// TIA Portal V18 export
ORGANIZATION_BLOCK "Main"   // OB1, LAD, ProgramCycle
TITLE = "Main Program Sweep (Cycle)"
{ S7_Optimized_Access := 'TRUE' }
// Bonanza Elect TD Rev0
// Written By Kristopher Gimenez January 16,2023
// For any questions please contact Automated Rig Technogies @ 403-723-6602
// This program is for the control the Bonanza Top drives utlizing the electric HPU.
// stored: SetENOAutomatically false
   VAR_INPUT
      Initial_Call : Bool;   // Initial call of this OB
      Remanence : Bool;   // =True, if remanent data are available
   END_VAR
   VAR_TEMP   // added for the SCL form of the ladder/FBD networks
      _w1 : Bool;
   END_VAR
BEGIN

REGION Network 2: Comm Checks, Communication is online after control system is powered up for 1min 10s. So to check when the system is full powered up
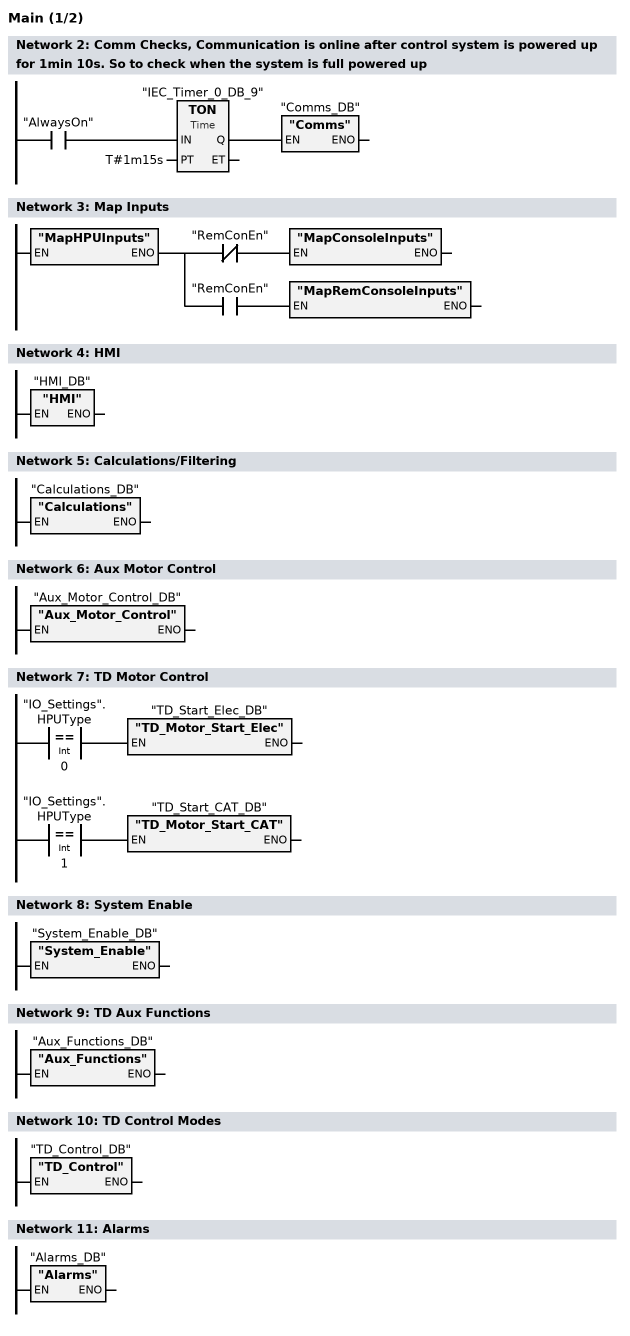
   RUNG wire#powerrail
      Contact( "AlwaysOn" )
      { S7_Templates := "time_type := Time" } "IEC_Timer_0_DB_9".TON(pt := T#1m15s, et =>)
      "Comms_DB"()
   END_RUNG
   // the same network as SCL:
   "IEC_Timer_0_DB_9".TON(IN := "AlwaysOn", PT := T#1m15s);
   IF "IEC_Timer_0_DB_9".Q THEN
       "Comms_DB"();   // "Comms"
   END_IF;
END_REGION

REGION Network 3: Map Inputs
   RUNG wire#powerrail
      "MapHPUInputs"()
      wire#w1
      I_Contact( "RemConEn" )
      "MapConsoleInputs"()
   END_RUNG
   RUNG wire#w1
      Contact( "RemConEn" )
      "MapRemConsoleInputs"()
   END_RUNG
   // the same network as SCL:
   "MapHPUInputs"(ENO => #_w1);
   IF #_w1 AND NOT "RemConEn" THEN "MapConsoleInputs"(); END_IF;
   IF #_w1 AND "RemConEn" THEN "MapRemConsoleInputs"(); END_IF;
END_REGION

REGION Network 4: HMI
   RUNG wire#powerrail
      "HMI_DB"()
   END_RUNG
   // the same network as SCL:
   "HMI_DB"();   // "HMI"
END_REGION

REGION Network 5: Calculations/Filtering
   RUNG wire#powerrail
      "Calculations_DB"()
   END_RUNG
   // the same network as SCL:
   "Calculations_DB"();   // "Calculations"
END_REGION

REGION Network 6: Aux Motor Control
   RUNG wire#powerrail
      "Aux_Motor_Control_DB"()
   END_RUNG
   // the same network as SCL:
   "Aux_Motor_Control_DB"();   // "Aux_Motor_Control"
END_REGION

REGION Network 7: TD Motor Control
   RUNG wire#powerrail
      { S7_Templates := "SrcType := Int" } EQ_Contact(in1 := "IO_Settings".HPUType, in2 := 0)
      "TD_Start_Elec_DB"()
   END_RUNG
   RUNG wire#powerrail
      { S7_Templates := "SrcType := Int" } EQ_Contact(in1 := "IO_Settings".HPUType, in2 := 1)
      "TD_Start_CAT_DB"()
   END_RUNG
   // the same network as SCL:
   IF "IO_Settings".HPUType = 0 THEN
       "TD_Start_Elec_DB"();   // "TD_Motor_Start_Elec"
   END_IF;
   IF "IO_Settings".HPUType = 1 THEN
       "TD_Start_CAT_DB"();   // "TD_Motor_Start_CAT"
   END_IF;
END_REGION

REGION Network 8: System Enable
   RUNG wire#powerrail
      "System_Enable_DB"()
   END_RUNG
   // the same network as SCL:
   "System_Enable_DB"();   // "System_Enable"
END_REGION

REGION Network 9: TD Aux Functions
   RUNG wire#powerrail
      "Aux_Functions_DB"()
   END_RUNG
   // the same network as SCL:
   "Aux_Functions_DB"();   // "Aux_Functions"
END_REGION

REGION Network 10: TD Control Modes
   RUNG wire#powerrail
      "TD_Control_DB"()
   END_RUNG
   // the same network as SCL:
   "TD_Control_DB"();   // "TD_Control"
END_REGION

REGION Network 11: Alarms
   RUNG wire#powerrail
      "Alarms_DB"()
   END_RUNG
   // the same network as SCL:
   "Alarms_DB"();   // "Alarms"
END_REGION

REGION Network 12: Indicators
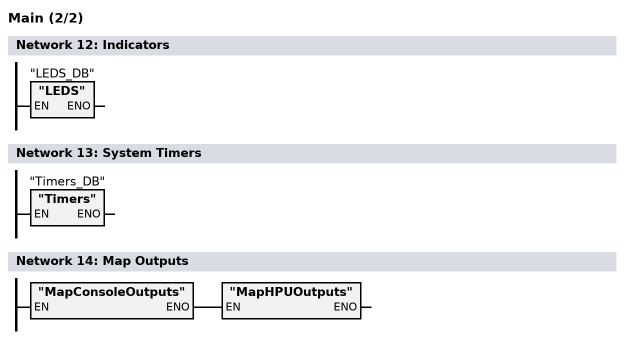
   RUNG wire#powerrail
      "LEDS_DB"()
   END_RUNG
   // the same network as SCL:
   "LEDS_DB"();   // "LEDS"
END_REGION

REGION Network 13: System Timers
   RUNG wire#powerrail
      "Timers_DB"()
   END_RUNG
   // the same network as SCL:
   "Timers_DB"();   // "Timers"
END_REGION

REGION Network 14: Map Outputs
   RUNG wire#powerrail
      "MapConsoleOutputs"()
      "MapHPUOutputs"()
   END_RUNG
   // the same network as SCL:
   "MapConsoleOutputs"(ENO => #_w1);
   IF #_w1 THEN "MapHPUOutputs"(); END_IF;
END_REGION
END_ORGANIZATION_BLOCK
